// TIA Portal V20 export
TYPE "typeEm5MonitoringJobInterface"
// stored: Access Published, Namespace Unit1
   STRUCT
      busyManPpUnloading { ExternalWritable := 'False'} : Bool;
      doneManPpUnloading { ExternalWritable := 'False'} : Bool;
   END_STRUCT;
END_TYPE
